// TIA Portal V17 export
// export: Created 2025-03-05T08:02:16.7397346Z, ExportSetting WithDefaults, DisplayName Totally Integrated Automation Portal, DisplayVersion V17 Update 8, DisplayName TIA Portal Openness, DisplayVersion V17 Update 8, DisplayName TIA Portal Version Control Interface, DisplayVersion V17, DisplayName SINAMICS Startdrive Advanced, DisplayVersion V17 SP2, DisplayName SINAMICS Startdrive G110M, G120, G120C, G120D, G120P, G115D, DisplayVersion V17 SP2, DisplayName SINAMICS Startdrive G130, G150, S120, S150, SINAMICS MV, S210, DisplayVersion V17 SP2, DisplayName STEP 7 Professional, DisplayVersion V17 Update 8, DisplayName SINUMERIK ONE STEP 7 Toolbox, DisplayVersion V17 Update 12, DisplayName SINUMERIK 840D sl STEP 7 Toolbox, DisplayVersion V17 Update 12, DisplayName STEP 7 Safety, DisplayVersion V17 Update 6, DisplayName WinCC Advanced, DisplayVersion V17 Update 8
TYPE "BA_MODE"
// stored: IsFailsafeCompliant false
   STRUCT
      BA1_INPUT : Bool;   // BA1 MODE INPUT
      BA2_INPUT : Bool;   // BA2 MODE INPUT
      BA3_INPUT : Bool;   // BA3 MODE INPUT
      BA5_INPUT : Bool;   // BA5 MODE INPUT
      CHANGE_ENABLE_INPUT : Bool;   // CHANGE ENABLE INPUT / CHANGE MODE ENABLE INPUT
      CHANGE_GENERAL_CONDITONS : Bool;   // CHANGE GENERAL CONDITIONS / CHANGE MODE GENERAL CONDITIONS
      CHANGE_INITIAL_CONDITIONS : Bool;   // CHANGE INITIAL CONDITIONS / CHANGE MODE INITIAL CONDITIONS
      BA1_REQUEST : Bool;   // MODE BA1 REQUEST / BA1 MODE REQUEST
      BA2_REQUEST : Bool;   // MODE BA2 REQUEST / BA2 MODE REQUEST
      BA3_REQUEST : Bool;   // MODE BA3 REQUEST / BA3 MODE REQUEST
      BA5_REQUEST : Bool;   // MODE BA5 REQUEST / BA5 MODE REQUEST
      BA1_SELECTED : Bool;   // MODE BA1 SELECTED / BA1 MODE SELECTED
      BA2_SELECTED : Bool;   // MODE BA2 SELECTED / BA2 MODE SELECTED
      BA3_SELECTED : Bool;   // MODE BA3 SELECTED / BA3 MODE SELECTED
      BA5_SELECTED : Bool;   // MODE BA5 SELECTED / BA5 MODE SELECTED
      BA3_SAFE_ENABLED : Bool;   // MODE BA3 SAFETY ENABLED / BA3 MODE SAFE ENABLED
      NO_BA_SELECTED : Bool;   // NO MODE BA MODE SELECTED / NO BA MODE SELECTED
      BA1_DISABLE : Bool;   // BA1 MODE DISABLED / BA1 MODE DISABLE
      BA2_BA3_BA5_DISABLE : Bool;   // BA2-BA3-BA5 DISABLED / BA2 BA3 BA5 MODE DISABLE
      TIME_EXCEEDED_SELECTION_ALARM : Bool;   // TIME EXCEDED SELECTION FAULT / TIME EXCEEDED ALARM
      CHANGE_TO_BA1_ALARM : Bool;   // BA1 MODE SELECTION FAULT / CHANGE TO BA1 MODE ALARM
      CHANGE_TO_BA2_ALARM : Bool;   // BA2 MODE SELECTION FAULT / CHANGE TO BA2 MODE ALARM
      CHANGE_TO_BA3_ALARM : Bool;   // BA3 MODE SELECTION FAULT / CHANGE TO BA3 MODE ALARM
      CHANGE_TO_BA5_ALARM : Bool;   // BA5 MODE SELECTION FAULT / CHANGE TO BA5 MODE ALARM
      BA1_SELECTED_MEMORY : Bool;   // BA1 MODE SELECTION FAULT / BA1 MODE SELECTED MEMORY
      BA2_SELECTED_MEMORY : Bool;   // BA2 MODE SELECTION FAULT / BA2 MODE SELECTED MEMORY
      BA3_SELECTED_MEMORY : Bool;   // BA3 MODE SELECTION FAULT / BA3 MODE SELECTED MEMORY
      BA5_SELECTED_MEMORY : Bool;   // BA5 MODE SELECTION FAULT / BA5 MODE SELECTED MEMORY
      WARNING_GONE : Bool;   // BA5 MODE SELECTION FAULT / WARNING GONE
      CHANGE_GENERAL_CONDITONS_HELP : Bool;   // CHANGE GENERAL CONDITIONS / CHANGE MODE GENERAL CONDITIONS HELP
      CHANGE_INITIAL_CONDITIONS_HELP : Bool;   // CHANGE INITIAL CONDITIONS / CHANGE MODE INITIAL CONDITIONS HELP
      TIMER_BA3 : TON_TIME;   // BA3 MODE TIMER
   END_STRUCT;
   // TIMER_BA3.PT := T#2s;
END_TYPE
